(* CoDeSys 2.3.9.50 project: 2D.pr6 *)
(* Libraries: STANDARD.LB6 5.6.98 12:03:02 *)

(* POU MAIN, LD *)
PROGRAM MAIN
VAR
	Stop AT %IX0.1: BOOL;
	GO2 AT %IX0.1: BOOL;
	GO1 AT %IX0.0: BOOL;
	Motor AT %QX0.0: BOOL;
	Light AT %QX0.0: BOOL;
END_VAR
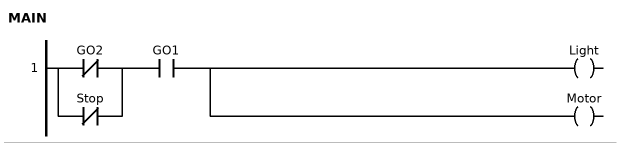
_LD_ (* Ladder Diagram *)
NETWORK 1
	{ [/GO2] | [/Stop] } - [GO1] --- (Light) (Motor)
_END_LD_
(* the same logic as Structured Text *)
(* Network 1 *)
Light := (NOT GO2 OR NOT Stop) AND GO1;
Motor := Light;
END_PROGRAM
